PROGRAM Dosificador_Polvo_1
VAR
	fbDosificador_P1 :Equipo_Motor_ATV320;
	Balanza_P1_WT1: Balanza;
	fbTR_P1_VI: Equipo_Motor_ATV320;
	TararP1:BOOL;
	dHS:DINT;
	
	Tmr_Alr_ZeroSpeed: TON;
	TDemoraInyectarPolvo: TON;
	Tiempo_seg_to_TIME_TDemoraInyec: Tiempo_seg_to_TIME;
	Auxtdemora: TIME;
	Calc_Veloc_Polvo_1: Calc_Veloc_Polvo;
	Calc_Veloc_Polvo_1i: Calc_Veloc_Polvo;
	Tiempo_seg_to_TIME_TInyeccion: Tiempo_seg_to_TIME;
	AuxInyec: TIME;
	TInyeccion: TON;
	ModoCalibrarP1 :BOOL;
	
	InyectarCalibrarP1: BOOL;
	Calibracion_Po_calc_P1: Calibracion_Po_calc;
	PolvoAsociado:STRING;
	TR_P1_WT1_rValue_REAL: REAL;
	TON_SolicitaPo: TON;
END_VAR
VAR PERSISTENT
	UltimaCalibracao	:UDINT;	//Data da ultima calibração feita com sucesso
END_VAR
VAR // added by the converter: edge detectors and wires of the graphical bodies
    _w1, _w2, _w3 : BOOL;
    _ft1 : F_TRIG;
    _rt1 : R_TRIG;
END_VAR

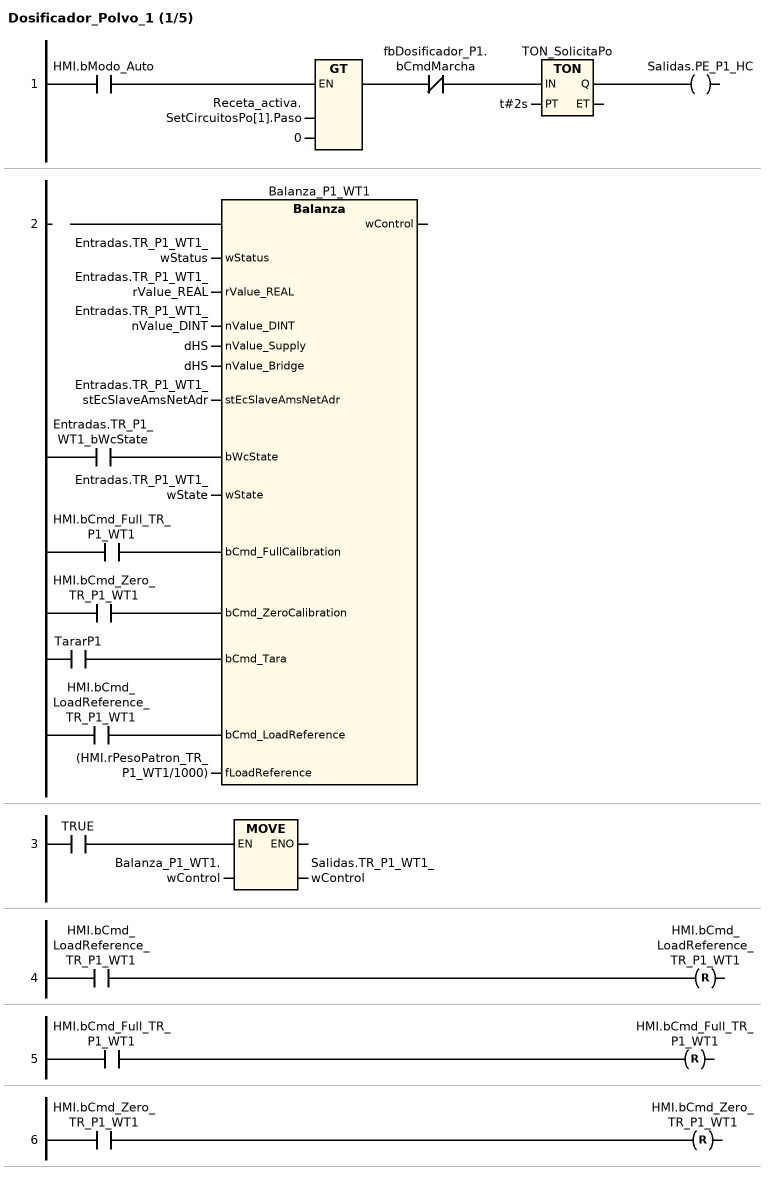
// NETWORK 1
TON_SolicitaPo(IN := (HMI.bModo_Auto AND Receta_activa.SetCircuitosPo[1].Paso > 0) AND NOT fbDosificador_P1.bCmdMarcha, PT := t#2s); // TON
Salidas.PE_P1_HC := TON_SolicitaPo.Q;

// NETWORK 2
Balanza_P1_WT1(
    wStatus := Entradas.TR_P1_WT1_wStatus,
    rValue_REAL := Entradas.TR_P1_WT1_rValue_REAL,
    nValue_DINT := Entradas.TR_P1_WT1_nValue_DINT,
    nValue_Supply := dHS,
    nValue_Bridge := dHS,
    stEcSlaveAmsNetAdr := Entradas.TR_P1_WT1_stEcSlaveAmsNetAdr,
    bWcState := Entradas.TR_P1_WT1_bWcState,
    wState := Entradas.TR_P1_WT1_wState,
    bCmd_FullCalibration := HMI.bCmd_Full_TR_P1_WT1,
    bCmd_ZeroCalibration := HMI.bCmd_Zero_TR_P1_WT1,
    bCmd_Tara := TararP1,
    bCmd_LoadReference := HMI.bCmd_LoadReference_TR_P1_WT1,
    fLoadReference := (HMI.rPesoPatron_TR_P1_WT1/1000)); // Balanza

// NETWORK 3
Salidas.TR_P1_WT1_wControl := Balanza_P1_WT1.wControl;

// NETWORK 4
HMI.bCmd_LoadReference_TR_P1_WT1 R= HMI.bCmd_LoadReference_TR_P1_WT1;

// NETWORK 5
HMI.bCmd_Full_TR_P1_WT1 R= HMI.bCmd_Full_TR_P1_WT1;

// NETWORK 6
HMI.bCmd_Zero_TR_P1_WT1 R= HMI.bCmd_Zero_TR_P1_WT1;

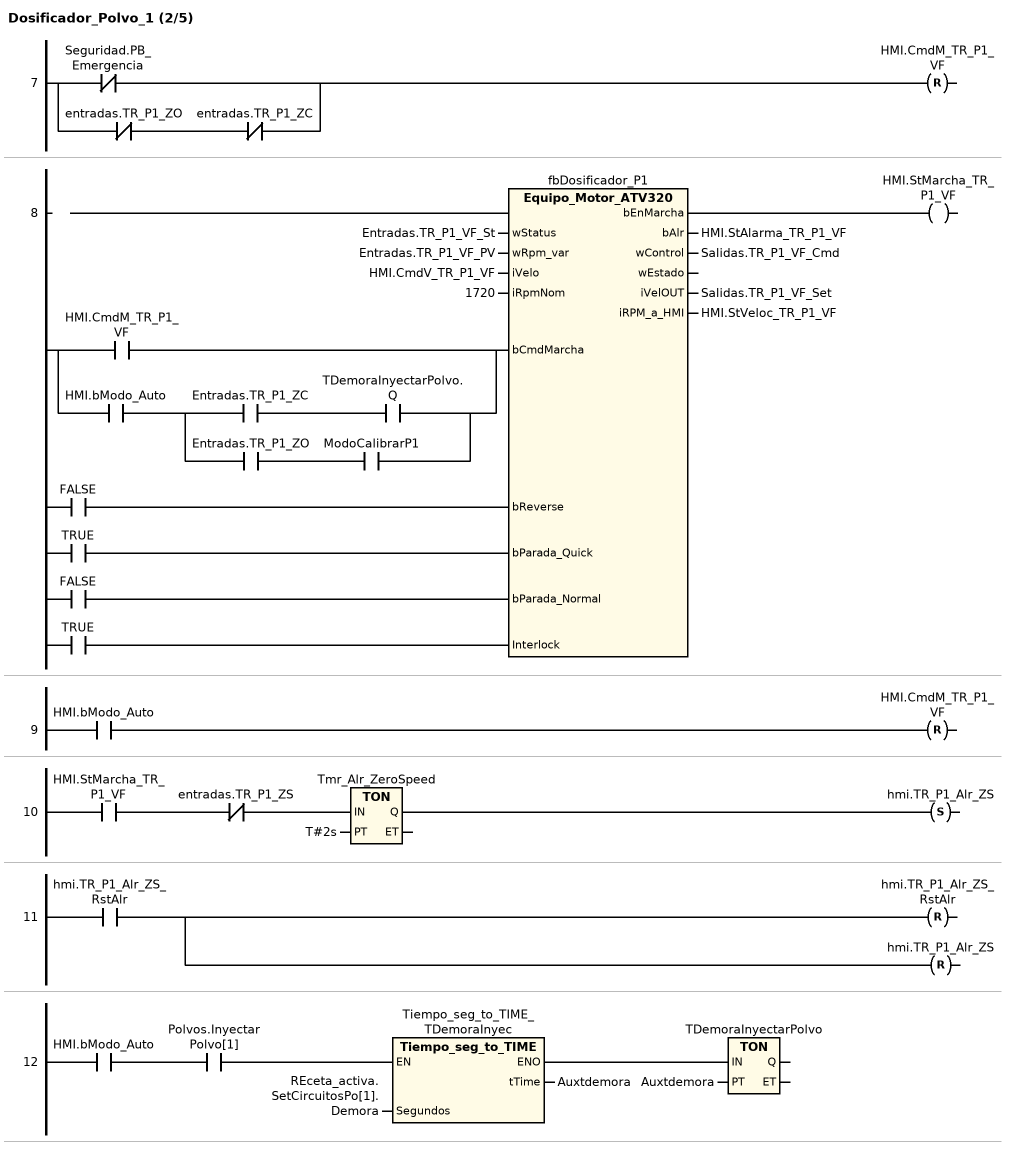
// NETWORK 7
HMI.CmdM_TR_P1_VF R= NOT Seguridad.PB_Emergencia OR NOT entradas.TR_P1_ZO AND NOT entradas.TR_P1_ZC;

// NETWORK 8
fbDosificador_P1(
    wStatus := Entradas.TR_P1_VF_St,
    wRpm_var := Entradas.TR_P1_VF_PV,
    iVelo := HMI.CmdV_TR_P1_VF,
    iRpmNom := 1720,
    bCmdMarcha := HMI.CmdM_TR_P1_VF OR HMI.bModo_Auto AND (Entradas.TR_P1_ZC AND TDemoraInyectarPolvo.Q OR Entradas.TR_P1_ZO AND ModoCalibrarP1),
    bReverse := FALSE,
    bParada_Quick := TRUE,
    bParada_Normal := FALSE,
    Interlock := TRUE,
    bAlr => HMI.StAlarma_TR_P1_VF,
    wControl => Salidas.TR_P1_VF_Cmd,
    iVelOUT => Salidas.TR_P1_VF_Set,
    iRPM_a_HMI => HMI.StVeloc_TR_P1_VF); // Equipo_Motor_ATV320
HMI.StMarcha_TR_P1_VF := fbDosificador_P1.bEnMarcha;

// NETWORK 9
HMI.CmdM_TR_P1_VF R= HMI.bModo_Auto;

// NETWORK 10
Tmr_Alr_ZeroSpeed(IN := HMI.StMarcha_TR_P1_VF AND NOT entradas.TR_P1_ZS, PT := T#2s); // TON
hmi.TR_P1_Alr_ZS S= Tmr_Alr_ZeroSpeed.Q;

// NETWORK 11
_w1 := hmi.TR_P1_Alr_ZS_RstAlr;
hmi.TR_P1_Alr_ZS_RstAlr R= _w1;
hmi.TR_P1_Alr_ZS R= _w1;

// NETWORK 12
_w2 := HMI.bModo_Auto AND Polvos.InyectarPolvo[1];
IF _w2 THEN
    Tiempo_seg_to_TIME_TDemoraInyec(Segundos := REceta_activa.SetCircuitosPo[1].Demora, tTime => Auxtdemora); // Tiempo_seg_to_TIME
END_IF
TDemoraInyectarPolvo(IN := _w2, PT := Auxtdemora); // TON

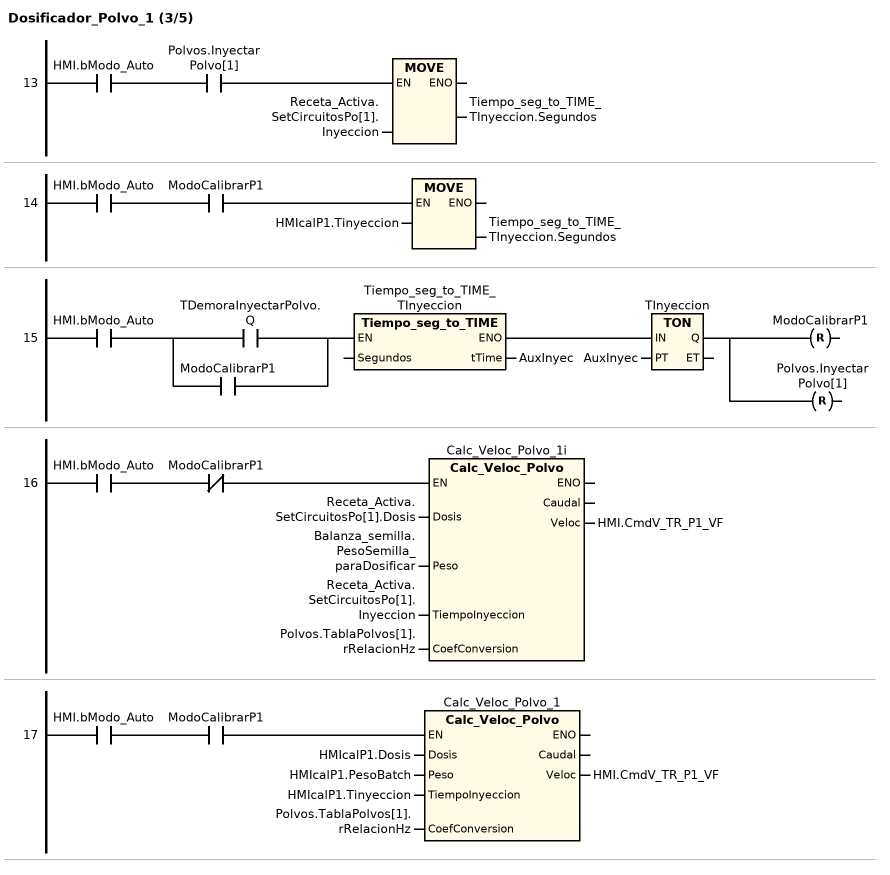
// NETWORK 13
IF HMI.bModo_Auto AND Polvos.InyectarPolvo[1] THEN
    Tiempo_seg_to_TIME_TInyeccion.Segundos := Receta_Activa.SetCircuitosPo[1].Inyeccion;
END_IF

// NETWORK 14
IF HMI.bModo_Auto AND ModoCalibrarP1 THEN Tiempo_seg_to_TIME_TInyeccion.Segundos := HMIcalP1.Tinyeccion; END_IF

// NETWORK 15
_w3 := HMI.bModo_Auto AND (TDemoraInyectarPolvo.Q OR ModoCalibrarP1);
IF _w3 THEN
    Tiempo_seg_to_TIME_TInyeccion(tTime => AuxInyec); // Tiempo_seg_to_TIME
END_IF
TInyeccion(IN := _w3, PT := AuxInyec); // TON
ModoCalibrarP1 R= TInyeccion.Q;
Polvos.InyectarPolvo[1] R= TInyeccion.Q;

// NETWORK 16
IF HMI.bModo_Auto AND NOT ModoCalibrarP1 THEN
    Calc_Veloc_Polvo_1i(
        Dosis := Receta_Activa.SetCircuitosPo[1].Dosis,
        Peso := Balanza_semilla.PesoSemilla_paraDosificar,
        TiempoInyeccion := Receta_Activa.SetCircuitosPo[1].Inyeccion,
        CoefConversion := Polvos.TablaPolvos[1].rRelacionHz,
        Veloc => HMI.CmdV_TR_P1_VF); // Calc_Veloc_Polvo
END_IF

// NETWORK 17
IF HMI.bModo_Auto AND ModoCalibrarP1 THEN
    Calc_Veloc_Polvo_1(
        Dosis := HMIcalP1.Dosis,
        Peso := HMIcalP1.PesoBatch,
        TiempoInyeccion := HMIcalP1.Tinyeccion,
        CoefConversion := Polvos.TablaPolvos[1].rRelacionHz,
        Veloc => HMI.CmdV_TR_P1_VF); // Calc_Veloc_Polvo
END_IF

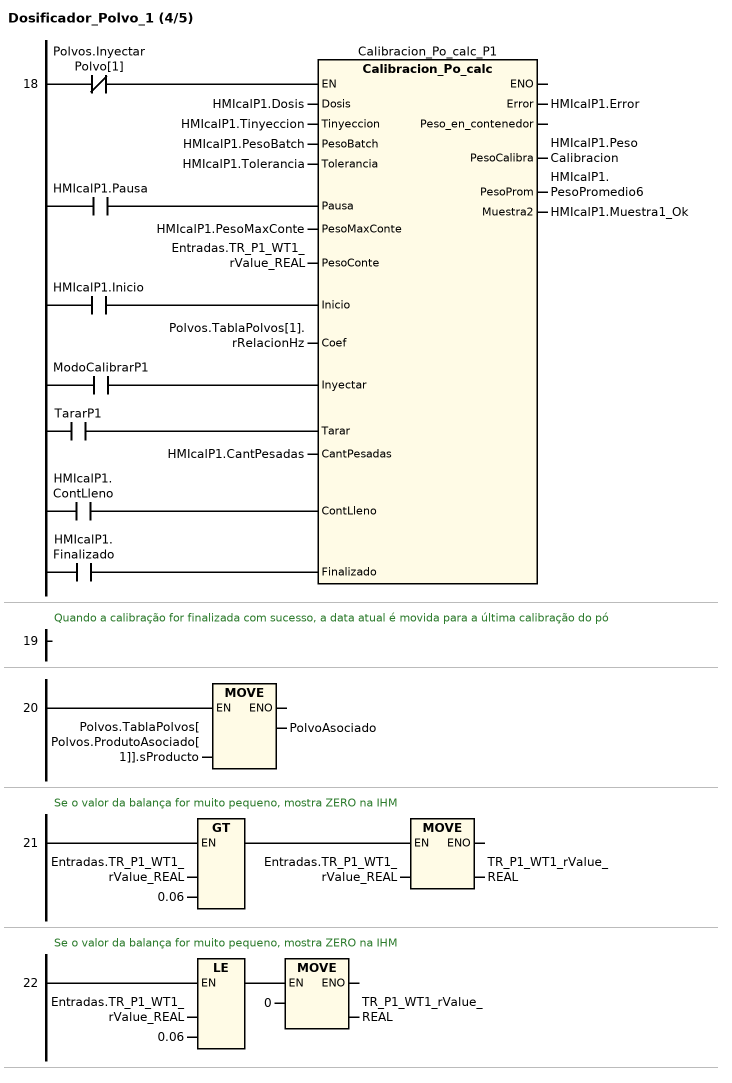
// NETWORK 18
IF NOT Polvos.InyectarPolvo[1] THEN
    Calibracion_Po_calc_P1(
        Dosis := HMIcalP1.Dosis,
        Tinyeccion := HMIcalP1.Tinyeccion,
        PesoBatch := HMIcalP1.PesoBatch,
        Tolerancia := HMIcalP1.Tolerancia,
        Pausa := HMIcalP1.Pausa,
        PesoMaxConte := HMIcalP1.PesoMaxConte,
        PesoConte := Entradas.TR_P1_WT1_rValue_REAL,
        Inicio := HMIcalP1.Inicio,
        Coef := Polvos.TablaPolvos[1].rRelacionHz,
        Inyectar := ModoCalibrarP1,
        Tarar := TararP1,
        CantPesadas := HMIcalP1.CantPesadas,
        ContLleno := HMIcalP1.ContLleno,
        Finalizado := HMIcalP1.Finalizado,
        Error => HMIcalP1.Error,
        PesoCalibra => HMIcalP1.PesoCalibracion,
        PesoProm => HMIcalP1.PesoPromedio6,
        Muestra2 => HMIcalP1.Muestra1_Ok); // Calibracion_Po_calc
END_IF

// NETWORK 19
// Quando a calibração for finalizada com sucesso, a data atual é movida para a última calibração do pó

// NETWORK 20
PolvoAsociado := Polvos.TablaPolvos[Polvos.ProdutoAsociado[1]].sProducto;

// NETWORK 21
// Se o valor da balança for muito pequeno, mostra ZERO na IHM
IF Entradas.TR_P1_WT1_rValue_REAL > 0.06 THEN TR_P1_WT1_rValue_REAL := Entradas.TR_P1_WT1_rValue_REAL; END_IF

// NETWORK 22
// Se o valor da balança for muito pequeno, mostra ZERO na IHM
IF Entradas.TR_P1_WT1_rValue_REAL <= 0.06 THEN TR_P1_WT1_rValue_REAL := 0; END_IF

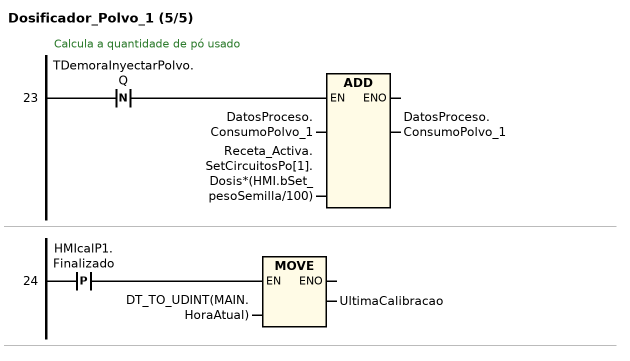
// NETWORK 23
// Calcula a quantidade de pó usado
_ft1(CLK := TDemoraInyectarPolvo.Q);
IF _ft1.Q THEN
    DatosProceso.ConsumoPolvo_1 := DatosProceso.ConsumoPolvo_1 + (Receta_Activa.SetCircuitosPo[1].Dosis*(HMI.bSet_pesoSemilla/100));
END_IF

// NETWORK 24
_rt1(CLK := HMIcalP1.Finalizado);
IF _rt1.Q THEN UltimaCalibracao := DT_TO_UDINT(MAIN.HoraAtual); END_IF

END_PROGRAM

(* stored: Version 1.1.0.1, ProductVersion 3.1.4024.14
   POU Dosificador_Polvo_1: Id {26d4816a-1841-4de7-a5f4-e197e2ecd524}, SpecialFunc None *)
